# EPICS autosave request: aliveApp/Db/aliveMSGCalc_settings.req
file calcout_settings.req P=$(P)aliveCalcMSG
